FUNCTION_BLOCK L3_PartDesEncap (* Basic Function Block Type *)
  (* Standard: 61499-2; Description: This block is used to desencapsulate all the events and data, used to manage the manufacturing of part, from an adapter. *)
  (* Version 0.0, 2014-09-24, EQUEROL, UJI *)
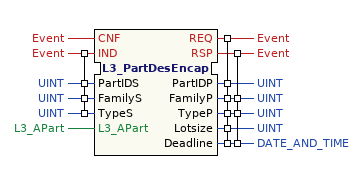
  EVENT_INPUT
    CNF; (* Normal Execution Request *)
    IND WITH PartIDS, FamilyS, TypeS; (* Ended part indication *)
  END_EVENT
  EVENT_OUTPUT
    REQ WITH PartIDP, FamilyP, TypeP, Lotsize, Deadline; (* Execution Confirmation *)
    RSP WITH FamilyP, TypeP, Deadline; (* Ended part reception confirmation *)
  END_EVENT
  VAR_INPUT
    PartIDS : UINT; (* Part identifier *)
    FamilyS : UINT; (* Part's family *)
    TypeS : UINT; (* Part's type *)
  END_VAR
  VAR_OUTPUT
    PartIDP : UINT; (* Identifier of the 1st part to be manufactured *)
    FamilyP : UINT; (* Part's family *)
    TypeP : UINT; (* Part's type *)
    Lotsize : UINT; (* Number of parts to be in the order *)
    Deadline : DATE_AND_TIME; (* Deadline of next part to be delivered *)
  END_VAR
  SOCKETS
    L3_APart : L3_APart;
  END_SOCKETS
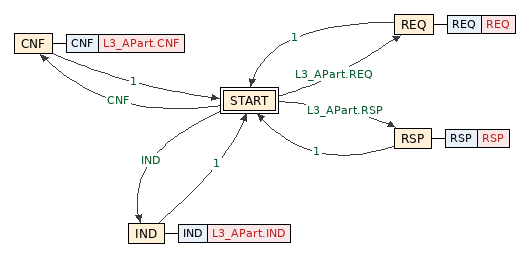
  EC_STATES
    START; (* Initial State *)
    REQ : REQ -> REQ; (* Normal execution *)
    RSP : RSP -> RSP;
    CNF : CNF -> L3_APart.CNF;
    IND : IND -> L3_APart.IND;
  END_STATES
  EC_TRANSITIONS
    START TO REQ := L3_APart.REQ;
    REQ TO START := 1;
    START TO RSP := L3_APart.RSP;
    RSP TO START := 1;
    START TO CNF := CNF;
    CNF TO START := 1;
    START TO IND := IND;
    IND TO START := 1;
  END_TRANSITIONS
  ALGORITHM REQ IN ST: (* Receives REQ event and data from the adapter *)
PartIDP := L3_APart.PartIDP;
FamilyP := L3_APart.FamilyP;
TypeP := L3_APart.TypeP;
Lotsize := L3_APart.Lotsize;
Deadline := L3_APart.Deadline;
  END_ALGORITHM
  ALGORITHM RSP IN ST: (* Receives RSPevent and data from the adapter *)
FamilyP := L3_APart.FamilyP;
TypeP := L3_APart.TypeP;
Deadline := L3_APart.Deadline;
  END_ALGORITHM
  ALGORITHM IND IN ST: (* Sends IND event and data through the adapter *)
L3_APart.PartIDS := PartIDS;
L3_APart.FamilyS := FamilyS;
L3_APart.TypeS := TypeS;
  END_ALGORITHM
  ALGORITHM CNF IN ST: (* Sends CNF event and data through the adapter *)
(*Nothing for now*)
  END_ALGORITHM
END_FUNCTION_BLOCK
